{attribute 'qualified_only'}
{attribute 'strict'}
TYPE E_ConvType :
(
	standard 	:= 0,
	end			:= 1,
	slave		:= 2
);
END_TYPE

(* stored: Version 1.1.0.1, ProductVersion 3.1.4024.4
   DUT E_ConvType: Id {ad520f9f-8d7c-42d1-9b8e-96f51edfe238} *)
